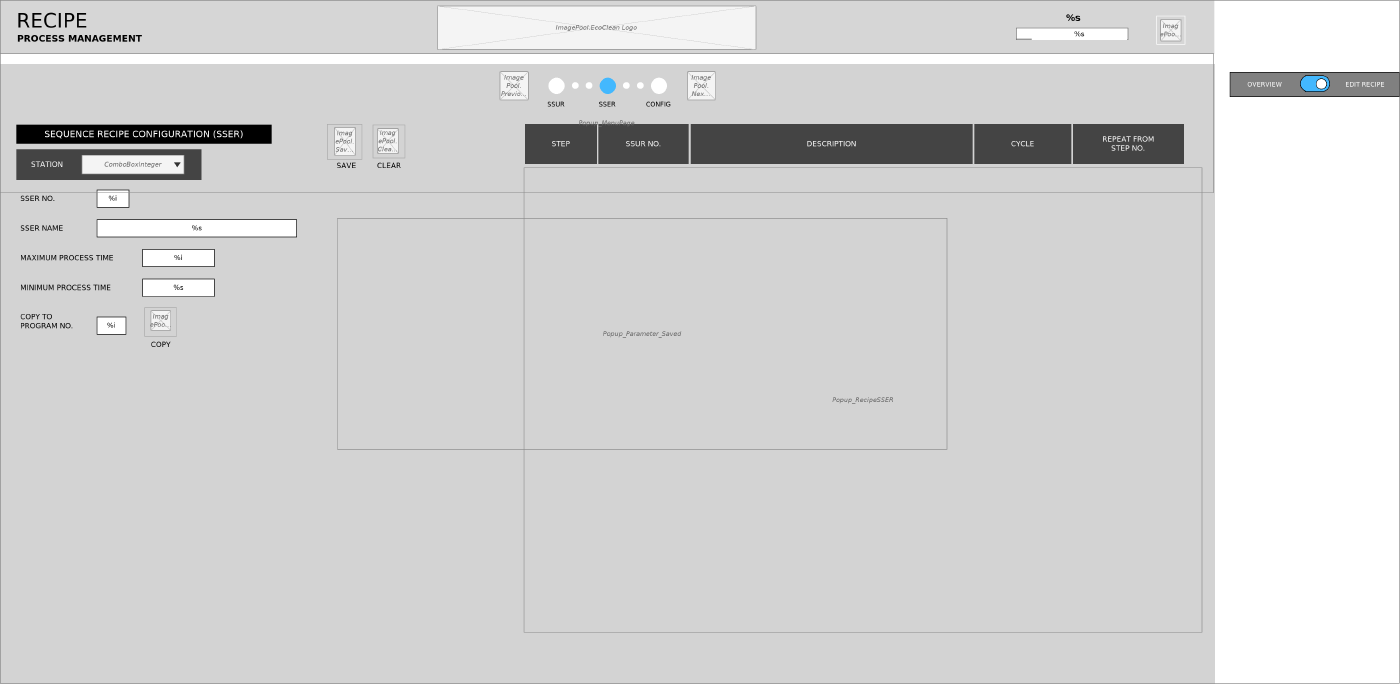
VISUALIZATION RecipeSSER_Page  // 2213x1082
    Rectangle (0,101 1920x981)
    Rectangle (0,63 1920x26)
        p3528305787: HMI_Ctrl.ANIMATION3
    Rectangle (0,0 1919x85)
    Group (23,6 321x67)
        Label (0,0 267x53), "RECIPE"
        Label (1,43 320x24), "PROCESS MANAGEMENT"
    Frame (828,265 1072x735)
        shows Popup_RecipeSSER()
    Rectangle (946,196 142x63), "SSUR NO."
    Rectangle (1092,196 445x63), "DESCRIPTION"
    Group (1828,25 45x45)
        OnMouseClick: toggle HMI_Ctrl.MenuButton
        RoundedRectangle (0,0 45x45), colour toggle: HMI_Ctrl.MenuButton
        Image (6,5 33x35), image: ImagePool.Menu Button
    Group (1944,113 269x41)
        RoundedRectangle (0,1 269x39)
        Label (1,0 108x41), "OVERVIEW"
        Label (161,0 105x41), "EDIT RECIPE"
        Group (111,6 47x26)
            OnMouseClick: change screen: Recipe_Page
            Group (0,0 47x26)
                Ellipse (0,0 26x26)
                Ellipse (21,0 26x26)
                RoundedRectangle (8,0 29x26)
            Ellipse (1,1 24x24)
            Ellipse (23,1 23x24)
            RoundedRectangle (9,1 28x24)
            Ellipse (25,5 17x17)
    Group (790,113 341x64)
        Ellipse (77,10 25x25)
        Ellipse (158,10 25x25)
        Ellipse (114,17 10x10)
        Ellipse (136,17 10x10)
        Ellipse (195,17 10x10)
        Ellipse (217,17 10x10)
        Ellipse (239,10 25x25)
        Label (57,40 64x24), "SSUR"
        Label (138,40 64x24), "SSER"
        Label (219,40 64x24), "CONFIG"
        Image (296,0 45x45), image: ImagePool.Next Button
            OnMouseClick: change screen: RecipeConfiguration_Page
        Image (0,0 45x45), image: ImagePool.Previous Button
            OnMouseClick: change screen: RecipeSSUR_Page
    Rectangle (26,197 403x30), "SEQUENCE RECIPE CONFIGURATION (SSER)"
    RoundedRectangle (26,236 292x48)
    Label (46,248 79x24), "STATION"
    ComboBoxInteger (129,245 162x30), variable: iStationNo, text list: 'TextList_Recipe'
    Label (29,302 93x24), "SSER NO."
    RoundedRectangle (153,300 51x28), "%i", text variable: DSScrMapSSER.iStationSequenceRecipeNo
        OnMouseDown: write the text variable via VisuDialogs.Numpad, min 1, max 20
    Label (29,396 174x24), "MAXIMUM PROCESS TIME"
    RoundedRectangle (225,394 114x28), "%i", text variable: DSScrMapSSER.DsStationSequenceRecipeMemory.iProcessMaxTime
        OnMouseDown: write the text variable via VisuDialogs.Numpad, min 1, max 9999
    Label (29,443 174x24), "MINIMUM PROCESS TIME"
    RoundedRectangle (225,441 114x28), "%s", text variable: DSScrMapSSER.DsStationSequenceRecipeMemory.iProcessMinTime
        OnMouseDown: write the text variable via VisuDialogs.Numpad, min 1, max 9999
    Label (29,349 101x24), "SSER NAME"
    RoundedRectangle (153,347 316x28), "%s", text variable: DSScrMapSSER.sStationSequenceRecipeDescription
        OnMouseDown: write the text variable via VisuDialogs.Keypad
    Label (29,488 110x41), "COPY TO PROGRAM NO."
    RoundedRectangle (153,501 46x28), "%i", text variable: DSScrMapSSER.iCopyToSubRecipeNo
        OnMouseDown: write the text variable via VisuDialogs.Numpad, min 1, max 20
    Rectangle (830,196 113x63), "STEP"
    Image (691,9 504x69), image: ImagePool.EcoClean Logo
    Rectangle (1540,196 153x63), "CYCLE"
    Rectangle (1696,196 175x63), "REPEAT FROM STEP NO."
    Group (228,486 51x71), invisible if: bMainOnOff
        Label (5,47 42x24), "COPY"
        RoundedRectangle (0,0 51x46), colour toggle: DSScrMapSSER.bCopyPB
            tap DSScrMapSSER.bCopyPB
        Image (10,5 32x32), image: ImagePool.Copy Button
            OnMouseDown: execute { DSScrMapSSER.bCopyPB:=1; }
            OnMouseUp: execute { DSScrMapSSER.bCopyPB:=0; }
    Group (1606,17 179x46)
        Button (0,27 177x19), image: VisuSymbols.Symbols.AddUser
        Rectangle (25,28 150x18), "%s", text variable: fbHmiTF1800_UserlevelManagement.dsHmiUserStatus_Active.sLoginName
        Rectangle (2,0 177x22), "%s", text variable: DSLocalSystemTimeML.sCurrentDT24Hr_General
    Group (517,196 56x80), invisible if: bMainOnOff
        Label (5,52 51x28), "SAVE", invisible if: bMainOnOff
        RoundedRectangle (0,0 55x56), colour toggle: bRecipeSavePb
            tap bRecipeSavePb
        Image (11,5 34x45), image: ImagePool.Save Button
            OnMouseDown: execute { bRecipeSavePb:=1; }
            OnMouseUp: execute { bRecipeSavePb:=0; }
    Frame (533,345 964x366), invisible if: NOT stWritePersistentData.SaveHR
        shows Popup_Parameter_Saved()
    Label (585,250 60x24), "CLEAR"
    RoundedRectangle (589,197 51x53), colour toggle: bRecipeClearInd_SSER
        tap bBufferClearPB_SSER[iStationNo]
    Image (596,203 34x40), image: ImagePool.Clear Button
        OnMouseDown: execute { bBufferClearPB_SSER[iStationNo]:=1; }
        OnMouseUp: execute { bBufferClearPB_SSER[iStationNo]:=0; }
    Frame (0,84 1918x221), invisible if: HMI_Ctrl.CloseMenuButton
        shows Popup_MenuPage()
END_VISUALIZATION

(* stored: Version 1.1.0.1, ProductVersion 3.1.4024.12
   Visu RecipeSSER_Page: Id {114d2c22-c408-42d1-bf86-0bdd3a618340} *)
